FUNCTION_BLOCK DIO_OUT (* Service Interface Function Block Type *)
  (* Standard: 61499-2 *)
  (* Version 0.0, 05/07/2021, josef, nxtControl GmBH, template *)
  PACKAGE Flexbridge.Iceblock;
  (* Compiler Cpp nxtControl builtin 1.0 *)
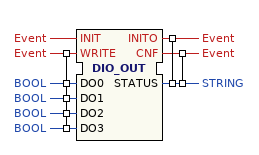
  EVENT_INPUT
    INIT;
    WRITE WITH DO0, DO1, DO2, DO3;
  END_EVENT
  EVENT_OUTPUT
    INITO WITH STATUS;
    CNF WITH STATUS;
  END_EVENT
  VAR_INPUT
    DO0 : BOOL := FALSE;
    DO1 : BOOL := FALSE;
    DO2 : BOOL := FALSE;
    DO3 : BOOL := FALSE;
  END_VAR
  VAR_OUTPUT
    STATUS : STRING;
  END_VAR
  SERVICE DIO_OUT/RESOURCE
    SEQUENCE normal_establishment
      DIO_OUT.INIT+(PARAMS) -> RESOURCE.initialize(PARAMS) -> DIO_OUT.INITO+();
    END_SEQUENCE
    SEQUENCE unsuccessful_establishment
      DIO_OUT.INIT+(PARAMS) -> RESOURCE.initialize(PARAMS) -> DIO_OUT.INITO-(STATUS);
    END_SEQUENCE
    SEQUENCE request_confirm
      DIO_OUT.REQ+(SD) -> RESOURCE.request(SD) -> DIO_OUT.CNF+(RD);
    END_SEQUENCE
    SEQUENCE request_inhibited
      DIO_OUT.REQ-(SD) -> DIO_OUT.CNF-(STATUS);
    END_SEQUENCE
    SEQUENCE request_error
      DIO_OUT.REQ+(SD) -> RESOURCE.request(SD) -> DIO_OUT.CNF-(STATUS);
    END_SEQUENCE
    SEQUENCE indication_response
      RESOURCE.indicate(RD) -> DIO_OUT.IND+(RD);
      DIO_OUT.RSP(QI,SD) -> RESOURCE.response(QI,SD);
    END_SEQUENCE
    SEQUENCE indication_inhibited
      RESOURCE.indicate(RD,QI=FALSE) -> RESOURCE.inhibited();
    END_SEQUENCE
    SEQUENCE error_indication
      RESOURCE.error(STATUS) -> DIO_OUT.IND-(STATUS);
    END_SEQUENCE
    SEQUENCE application_initiated_termination
      DIO_OUT.INIT-() -> RESOURCE.terminate() -> DIO_OUT.INITO-(STATUS);
    END_SEQUENCE
    SEQUENCE resource_initiated_termination
      -> DIO_OUT.INITO-(STATUS);
    END_SEQUENCE
  END_SERVICE
END_FUNCTION_BLOCK
